# B&R Automation Studio project FileXplore
Automation Studio 6.7.0.187; technology packages: mappCockpit 6.6.0, mappView 6.6.0, OpcUaCs 6.6.1

## Configuration PLC

CPU X20CP3687X, AutomationRuntime 6.8.1, Build 11.3.0, Vc 6.0.0

### Task classes (Cpu.sw)
```
Cyclic#1:
  XFiles <- Source.XFiles.prg
Binaries: FWRules, ArSvcReg, TCData, udbdef, TCLang, mvLoader, mvConfig, User, iomap, TC, sysconf, BRRole, Role, arconfig, asfw, ashwac, Settings, UaCsConfig, ashwd, mCoWebSc
Libraries: runtime, AsZip, FileIO, AsHttp, UaCore, UaCoal, AsIecCon, ArSsl, UaCoalPrv, CoTrace, XFileLib, AsIODiag
```

### Hardware
```
X20CP3687X : X20CP3687X v1.9.0.0
  Connector IF2:
    ActivateDevice = 1
    Mode = Manual
    InternetAddress = 192.168.3.100
    SubnetMask = 255.255.255.0
    ActivateSnmp = 2
  ConfigurationID = FileXplore_PLC
  UserPartitionSize = 100
  Simulation = 1
  FileDevice1
  FileDeviceName1 = USER
  FileDevicePath1 = USER_PATH
  FileDevice2
  FileDeviceName2 = XPlore
  FileDevicePath2 = USER_PATH\XPlore
  ActivateFtpServer = 1
  FTPProtocol = 1
  FtpUser1
  FtpUsername1 = FileX
  FtpUserPassword1 = 8JF6nSqDfWDJ2i1aTp85XN0mfqkVcSXatZ/FMR942Jg=  // Password: XFile
  FtpUserSalt1 = RJsmGuSw
  FTPAccessRight1 = 0
  ActivateWebServer = 1
  WebServerProtocol = 3
  HttpsSslCfg = SSLConfiguration
  WebServerWebDir = dist\
```

## Logical view

Binary libraries used (declarations not repeated): operator, runtime, AsIecCon, AsZip, FileIO, AsHttp, CoTrace 6.5.0, AsIODiag

### Global.var - Global variables
```iecst
VAR
	gHostIP : STRING[15];
END_VAR
```


### Package Logical/FileXplore - File Xplorer source code (vite/react)

### CHANGELOG.md
```markdown
# Changelog

All notable changes to FileXplorer are documented here.

## [2.0.2] - 2026-10-08
- Added `ForceConvertToUTF8` config option: files whose extension is listed are converted to UTF-8 before transfer (BOM-aware, with Windows ANSI/CP1252 and UTF-16 fallback). An empty or missing list disables conversion.
- Added a Refresh button to reload the current folder without leaving it.
- Fixed the Home button doing nothing when already at the default path; it now always reloads.

## [2.0.1] - 2026-09-30
- FileXplore version shown only 1 second

## [2.0.0] - 2026-09-25

- Added a version display showing FileXplore for five seconds.
- Modified ftp to chunked HTTPS file uploads (works in arsim also)
- Added filename header sanitization for PLC-compatible transfers.
- Added configurable file browsing and transfer settings.
```

- package-lock.json (not shown)

- package.json (not shown)

### README.md
~~~~markdown
# File Explorer with HTTPS Transfer

A Vite + React file explorer application with Node.js backend designed for **B&R mappView environments**. The application enables browsing local files and transferring them to a PLC over chunked HTTPS, featuring real-time progress tracking and transfer recovery handling.

## Use Case

This application is intended to run in **B&R mappView** environments where:
- The **frontend** runs in the mappView HMI interface
- The **Node.js backend** runs on a **Panel PC** or another platform capable of accessing the local file system
- The **HTTPS endpoint** is a **B&R PLC** service that receives the selected files from the file explorer
- Files are streamed from the Panel PC (or host platform) to the PLC via bounded HTTPS chunks

## Features

### File Browsing
- Browse files and directories from configured drives on your local machine
- Tree-view navigation with expand/collapse folders
- Drive selection dropdown
- Configurable file extension filtering (e.g., `.txt`, `.cnc`)
- Access restrictions to prevent navigation outside configured directories

### HTTPS Transfer
- One-click file transfer to HTTPS endpoint (B&R PLC)
- Real-time upload progress tracking using Server-Sent Events (SSE)
- Visual progress bar showing actual HTTPS transfer percentage
- Transfer cancellation support (client and server-side)
- Configurable chunk size, timeout, and retry handling for transient transfer failures
- Automatic file load command trigger after successful upload to PLC
- Green highlight for successfully transferred files

### Configuration
- **Frontend Config** (`public/config.json`): Supported file extensions and default drive paths
- **Backend Config** (`server/https-config.json`): PLC HTTPS endpoint, chunk size, timeout, retry, default folder, and filename settings

## Project Structure

```
├── public/
│   └── config.json          # Frontend configuration
├── server/
│   ├── index.js             # Express backend server
│   └── https-config.json    # HTTPS transfer configuration
├── src/
│   ├── App.jsx              # Main React application
│   ├── App.css              # Application styles
│   └── main.jsx             # React entry point
└── dist/                    # Production build output
```

## Getting Started

### Backend Server (Panel PC or Host Platform)
The Node.js backend should run on a Panel PC or any platform with access to the local file system containing the files to be transferred.

```bash
cd server
node index.js
```
Server runs on `http://localhost:5000`

### Frontend (mappView HMI)
For development:
```bash
npm run dev
```
Development server runs on `http://localhost:5173`

### Production Build (for mappView deployment)
```bash
npm run build
node serve-dist.js
```
Serves production build on `http://localhost:3000`

The `dist` folder can be deployed to the mappView project.

## Running Backend as a Windows Service

To ensure the Node.js backend server runs automatically on PC startup and restarts after reboots, set it up as a Windows service.

### Option 1: Using node-windows (Recommended)

1. Install node-windows in the server directory:
```bash
cd server
npm install node-windows
```

2. Create a service installation script `install-service.js`:
```javascript
const Service = require('node-windows').Service;
const path = require('path');

// Create a new service object
const svc = new Service({
  name: 'FileExplorer Backend',
  description: 'File Explorer Node.js backend for B&R mappView',
  script: path.join(__dirname, 'index.js'),
  nodeOptions: [
    '--harmony',
    '--max_old_space_size=4096'
  ]
});

// Listen for the "install" event
svc.on('install', function() {
  svc.start();
  console.log('Service installed and started!');
});

// Install the service
svc.install();
```

3. Run the installation script as Administrator:
```bash
node install-service.js
```

4. To uninstall the service, create `uninstall-service.js`:
```javascript
const Service = require('node-windows').Service;
const path = require('path');

const svc = new Service({
  name: 'FileExplorer Backend',
  script: path.join(__dirname, 'index.js')
});

svc.on('uninstall', function() {
  console.log('Service uninstalled');
});

svc.uninstall();
```

### Option 2: Using Windows Task Scheduler

1. Open Task Scheduler (taskschd.msc)
2. Click "Create Task" (not "Create Basic Task")
3. **General tab**:
   - Name: "FileExplorer Backend"
   - Select "Run whether user is logged on or not"
   - Check "Run with highest privileges"
4. **Triggers tab**:
   - New → Begin the task: "At startup"
   - Delay task for: 30 seconds (to ensure network is ready)
5. **Actions tab**:
   - New → Action: "Start a program"
   - Program/script: `C:\Program Files\nodejs\node.exe`
   - Add arguments: `C:\path\to\your\server\index.js`
   - Start in: `C:\path\to\your\server`
6. **Conditions tab**:
   - Uncheck "Start the task only if the computer is on AC power"
7. Click OK and enter your Windows password

### Option 3: Using PM2 (Alternative)

1. Install PM2 globally:
```bash
npm install -g pm2
npm install -g pm2-windows-startup
```

2. Configure PM2 to start on boot:
```bash
pm2-startup install
```

3. Start your application with PM2:
```bash
cd server
pm2 start index.js --name "fileexplorer-backend"
pm2 save
```

### Verify Service is Running

Check if the service is running by accessing `http://localhost:5000/api/drives` in a browser or test it after a reboot.

## API Endpoints

- `GET /api/drives` - List available drives on the host platform
- `GET /api/list?path=<path>` - List directory contents from host file system
- `GET /api/read-file?path=<path>` - Read file as binary stream from host
- `POST /api/save-to-https-static` - Stream file from backend host to PLC HTTPS endpoint in chunks with progress (SSE)
- `POST /api/cancel-upload` - Cancel active HTTPS upload to PLC
- `POST /api/load-selected-file` - Trigger file load command on PLC

## Technologies

- **Frontend**: React 18, Vite, CSS (deployable to B&R mappView HTML )
- **Backend**: Node.js, Express (runs on Panel PC or host platform)
- **Transfer**: Node.js native HTTPS chunk upload client
- **Progress Tracking**: Server-Sent Events (SSE)
- **Target**: B&R PLC with HTTPS service capability
~~~~

- config.json (not shown)

- ftp-config.json (not shown)

### How to run.txt
```
1. Install node.js server (Chrome downloads)
2. Install Express via npm install express (from command line)
3. Install the node production process manager and run the node application (from command line):
	npm install -g pm2
	pm2 start app.js
	pm2 save
	pm2-startup install
```

- https-config.json (not shown)

- package-lock.json (not shown)

- package.json (not shown)

- App.jsx (not shown)

### Package Logical/Source - Source code for PLC code

### Library Logical/Source/XFileLib (IEC) - Library for file managment backend functionality

#### Types.typ - Exported data types
```iecst
TYPE
	XploreUploadStep_typ :
		(
		XPLORE_UPLOAD_IDLE := 0,
		XPLORE_UPLOAD_DELETE := 10,
		XPLORE_UPLOAD_CREATE := 20,
		XPLORE_UPLOAD_OPEN := 30,
		XPLORE_UPLOAD_WRITE := 40,
		XPLORE_UPLOAD_CLOSE := 50,
		XPLORE_UPLOAD_RESPOND := 60,
		XPLORE_UPLOAD_ERROR := 100
		);
	XploreHttpsServices_typ : 	STRUCT
		LoadServiceName : STRING[80];
		UploadServiceName : STRING[80];
		FileDevice : STRING[20];
		LoadRequestHeader : httpRequestHeader_t;
		LoadRequest : STRING[1000];
		LoadResponseHeader : httpResponseHeader_t;
		LoadResponse : STRING[1000];
		UploadRequestHeader : httpRequestHeader_t;
		UploadData : ARRAY[0..MAX_DATA_PAYLOAD_SIZE_BYTES]OF USINT;
		UploadResponseHeader : httpResponseHeader_t;
		UploadResponse : STRING[1000];
		FileName : STRING[80];
		TransferId : STRING[80];
		UploadOffset : UDINT;
		UploadLength : UDINT;
		UploadFileSize : UDINT;
		UploadChunkIndex : UDINT;
		UploadBytesReceived : UDINT;
		UploadStep : XploreUploadStep_typ;
		FileIdent : UDINT;
		Busy : BOOL;
		Done : BOOL;
		Error : BOOL;
		LastError : UINT;
		LastErrorText : STRING[80];
		LastHttpStatus : UINT;
		LastChunkFinal : BOOL;
		Reset : BOOL;
	END_STRUCT;
END_TYPE
```

#### Constants.var - Exported constants
```iecst
VAR CONSTANT
	MAX_DATA_PAYLOAD_SIZE_BYTES : UDINT := 1048576*MAX_DATA_PAYLOAD_SIZE_MB;
	MAX_DATA_PAYLOAD_SIZE_MB : UDINT := 5; (*This is the value to set for the file transfer*)
END_VAR
```

#### XFileLib.fun - Exported functions and function blocks
```iecst
{REDUND_ERROR} {REDUND_UNREPLICABLE} FUNCTION_BLOCK XploreFileService (*Xplore file service (HTTPS)*) (*$GROUP=User,$CAT=User,$GROUPICON=User.png,$CATICON=User.png*)
	VAR_INPUT
		Enable : {REDUND_UNREPLICABLE} BOOL;
		Reset : {REDUND_UNREPLICABLE} BOOL;
		FileDevice : {REDUND_UNREPLICABLE} STRING[20];
		LoadServiceName : {REDUND_UNREPLICABLE} STRING[80];
		UploadServiceName : {REDUND_UNREPLICABLE} STRING[80];
	END_VAR
	VAR_OUTPUT
		Busy : {REDUND_UNREPLICABLE} BOOL;
		Done : {REDUND_UNREPLICABLE} BOOL;
		Error : {REDUND_UNREPLICABLE} BOOL;
		FileName : {REDUND_UNREPLICABLE} STRING[80];
		UploadBytesReceived : {REDUND_UNREPLICABLE} UDINT;
		LastError : {REDUND_UNREPLICABLE} UINT;
		LastErrorText : {REDUND_UNREPLICABLE} STRING[80];
		LastHttpStatus : {REDUND_UNREPLICABLE} UINT;
	END_VAR
	VAR
		loadHttpsService : {REDUND_UNREPLICABLE} httpsService;
		uploadHttpsService : {REDUND_UNREPLICABLE} httpsService;
		fileDelete : {REDUND_UNREPLICABLE} FileDelete;
		fileCreate : {REDUND_UNREPLICABLE} FileCreate;
		fileOpen : {REDUND_UNREPLICABLE} FileOpen;
		fileWrite : {REDUND_UNREPLICABLE} FileWrite;
		fileClose : {REDUND_UNREPLICABLE} FileClose;
		service : {REDUND_UNREPLICABLE} XploreHttpsServices_typ;
	END_VAR
END_FUNCTION_BLOCK
```

#### XploreFileService.st - Reusable XFiles HTTP and file transfer service
```iecst
FUNCTION_BLOCK XploreFileService
	service.LoadServiceName := LoadServiceName;
	service.UploadServiceName := UploadServiceName;
	service.FileDevice := FileDevice;

	loadHttpsService(enable := Enable AND NOT Reset,
		option := httpOPTION_SERVICE_TYPE_NAME,
		pServiceName := ADR(service.LoadServiceName),
		pRequestHeader := ADR(service.LoadRequestHeader),
		pRequestData := ADR(service.LoadRequest),
		requestDataSize := SIZEOF(service.LoadRequest),
		pResponseHeader := ADR(service.LoadResponseHeader),
		pResponseData := ADR(service.LoadResponse),
		responseDataLen := SIZEOF(service.LoadResponse));
	uploadHttpsService(enable := Enable AND NOT Reset,
		option := httpOPTION_SERVICE_TYPE_NAME,
		pServiceName := ADR(service.UploadServiceName),
		pRequestHeader := ADR(service.UploadRequestHeader),
		pRequestData := ADR(service.UploadData),
		requestDataSize := SIZEOF(service.UploadData),
		pResponseHeader := ADR(service.UploadResponseHeader),
		pResponseData := ADR(service.UploadResponse),
		responseDataLen := SIZEOF(service.UploadResponse));

	IF service.LoadRequestHeader.userLine[0].name = '' THEN
		service.LoadRequestHeader.userLine[0].name := 'fileName';
		service.UploadRequestHeader.userLine[0].name := 'fileName';
		service.UploadRequestHeader.userLine[1].name := 'remotePath';
		service.UploadRequestHeader.userLine[2].name := 'transferId';
		service.UploadRequestHeader.userLine[3].name := 'chunkOffset';
		service.UploadRequestHeader.userLine[4].name := 'chunkIndex';
		service.UploadRequestHeader.userLine[5].name := 'fileSize';
		service.UploadRequestHeader.userLine[6].name := 'finalChunk';
	END_IF

	IF loadHttpsService.phase = httpPHASE_RECEIVED THEN
		IF service.LoadRequest = 'Load' THEN
			service.LoadResponseHeader.status := '200 OK';
			service.LoadResponseHeader.contentType := 'text/plain';
			service.LoadResponse := 'Loading';
			service.LoadRequest := '';
			loadHttpsService.send := TRUE;
		END_IF
		service.FileName := service.LoadRequestHeader.userLine[0].value;
	ELSE
		loadHttpsService.send := FALSE;
	END_IF

	IF Reset OR NOT Enable THEN
		service.UploadStep := XPLORE_UPLOAD_IDLE;
		service.Busy := FALSE;
		service.Done := FALSE;
		service.Error := FALSE;
		service.LastError := ERR_OK;
		service.FileIdent := 0;
		uploadHttpsService.send := FALSE;
	ELSE
		IF (uploadHttpsService.phase = httpPHASE_RECEIVED) AND (service.UploadStep = XPLORE_UPLOAD_IDLE) THEN
			service.FileName := service.UploadRequestHeader.userLine[0].value;
			service.TransferId := service.UploadRequestHeader.userLine[2].value;
			service.UploadOffset := STRING_TO_UDINT(service.UploadRequestHeader.userLine[3].value);
			service.UploadChunkIndex := STRING_TO_UDINT(service.UploadRequestHeader.userLine[4].value);
			service.UploadFileSize := STRING_TO_UDINT(service.UploadRequestHeader.userLine[5].value);
			service.LastChunkFinal := service.UploadRequestHeader.userLine[6].value = '1';
			service.UploadLength := uploadHttpsService.requestDataLen;
			service.Busy := TRUE;
			service.Done := FALSE;
			service.Error := FALSE;
			service.LastError := ERR_OK;
			service.LastErrorText := '';
			service.LastHttpStatus := 0;
			IF uploadHttpsService.method <> httpMETHOD_POST THEN
				service.LastHttpStatus := 405;
				service.UploadStep := XPLORE_UPLOAD_ERROR;
			ELSIF service.FileName = '' THEN
				service.LastHttpStatus := 400;
				service.UploadStep := XPLORE_UPLOAD_ERROR;
			ELSIF service.UploadLength >= SIZEOF(service.UploadData) THEN
				service.LastHttpStatus := 413;
				service.UploadStep := XPLORE_UPLOAD_ERROR;
			ELSIF service.UploadOffset = 0 THEN
				service.UploadStep := XPLORE_UPLOAD_DELETE;
			ELSE
				service.UploadStep := XPLORE_UPLOAD_OPEN;
			END_IF
		END_IF

		CASE service.UploadStep OF
			XPLORE_UPLOAD_IDLE:
				uploadHttpsService.send := FALSE;

			XPLORE_UPLOAD_DELETE:
				fileDelete(enable := TRUE, pDevice := ADR(service.FileDevice), pName := ADR(service.FileName));
				IF (fileDelete.status = ERR_OK) OR (fileDelete.status = fiERR_FILE_NOT_FOUND) THEN
					fileDelete(enable := FALSE);
					service.UploadStep := XPLORE_UPLOAD_CREATE;
				ELSIF fileDelete.status <> ERR_FUB_BUSY THEN
					service.LastError := fileDelete.status;
					service.LastErrorText := UDINT_TO_STRING(UINT_TO_UDINT(fileDelete.status));
					service.LastHttpStatus := 500;
					fileDelete(enable := FALSE);
					service.UploadStep := XPLORE_UPLOAD_ERROR;
				END_IF

			XPLORE_UPLOAD_CREATE:
				fileCreate(enable := TRUE, pDevice := ADR(service.FileDevice), pFile := ADR(service.FileName));
				IF fileCreate.status = ERR_OK THEN
					service.FileIdent := fileCreate.ident;
					fileCreate(enable := FALSE);
					service.UploadStep := XPLORE_UPLOAD_WRITE;
				ELSIF fileCreate.status <> ERR_FUB_BUSY THEN
					service.LastError := fileCreate.status;
					service.LastErrorText := UDINT_TO_STRING(UINT_TO_UDINT(fileCreate.status));
					service.LastHttpStatus := 500;
					fileCreate(enable := FALSE);
					service.UploadStep := XPLORE_UPLOAD_ERROR;
				END_IF

			XPLORE_UPLOAD_OPEN:
				fileOpen(enable := TRUE, pDevice := ADR(service.FileDevice), pFile := ADR(service.FileName), mode := fiREAD_WRITE);
				IF fileOpen.status = ERR_OK THEN
					service.FileIdent := fileOpen.ident;
					fileOpen(enable := FALSE);
					service.UploadStep := XPLORE_UPLOAD_WRITE;
				ELSIF fileOpen.status <> ERR_FUB_BUSY THEN
					service.LastError := fileOpen.status;
					service.LastErrorText := UDINT_TO_STRING(UINT_TO_UDINT(fileOpen.status));
					service.LastHttpStatus := 409;
					fileOpen(enable := FALSE);
					service.UploadStep := XPLORE_UPLOAD_ERROR;
				END_IF

			XPLORE_UPLOAD_WRITE:
				fileWrite(enable := TRUE, ident := service.FileIdent, offset := service.UploadOffset, pSrc := ADR(service.UploadData), len := service.UploadLength);
				IF fileWrite.status = ERR_OK THEN
					fileWrite(enable := FALSE);
					service.UploadStep := XPLORE_UPLOAD_CLOSE;
				ELSIF fileWrite.status <> ERR_FUB_BUSY THEN
					service.LastError := fileWrite.status;
					service.LastErrorText := UDINT_TO_STRING(UINT_TO_UDINT(fileWrite.status));
					service.LastHttpStatus := 500;
					fileWrite(enable := FALSE);
					service.UploadStep := XPLORE_UPLOAD_CLOSE;
				END_IF

			XPLORE_UPLOAD_CLOSE:
				fileClose(enable := TRUE, ident := service.FileIdent);
				IF fileClose.status = ERR_OK THEN
					fileClose(enable := FALSE);
					service.FileIdent := 0;
					IF service.LastError = ERR_OK THEN
						service.UploadStep := XPLORE_UPLOAD_RESPOND;
					ELSE
						service.UploadStep := XPLORE_UPLOAD_ERROR;
					END_IF
				ELSIF fileClose.status <> ERR_FUB_BUSY THEN
					service.LastError := fileClose.status;
					service.LastErrorText := UDINT_TO_STRING(UINT_TO_UDINT(fileClose.status));
					service.LastHttpStatus := 500;
					fileClose(enable := FALSE);
					service.FileIdent := 0;
					service.UploadStep := XPLORE_UPLOAD_ERROR;
				END_IF

			XPLORE_UPLOAD_RESPOND:
				service.UploadBytesReceived := service.UploadOffset + service.UploadLength;
				service.UploadResponseHeader.status := '200 OK';
				service.UploadResponseHeader.contentType := 'text/plain';
				service.UploadResponse := 'OK';
				service.Done := service.LastChunkFinal;
				service.Busy := FALSE;
				uploadHttpsService.send := TRUE;
				service.UploadStep := XPLORE_UPLOAD_IDLE;

			XPLORE_UPLOAD_ERROR:
				service.Error := TRUE;
				service.Busy := FALSE;
				IF service.LastHttpStatus = 0 THEN
					service.LastHttpStatus := 500;
				END_IF
				IF service.LastHttpStatus = 400 THEN
					service.UploadResponseHeader.status := '400 Bad Request';
				ELSIF service.LastHttpStatus = 405 THEN
					service.UploadResponseHeader.status := '405 Method Not Allowed';
				ELSIF service.LastHttpStatus = 409 THEN
					service.UploadResponseHeader.status := '409 Conflict';
				ELSIF service.LastHttpStatus = 413 THEN
					service.UploadResponseHeader.status := '413 Payload Too Large';
				ELSE
					service.UploadResponseHeader.status := '500 Internal Server Error';
				END_IF
				service.UploadResponseHeader.contentType := 'text/plain';
				service.UploadResponse := service.LastErrorText;
				uploadHttpsService.send := TRUE;
				service.UploadStep := XPLORE_UPLOAD_IDLE;
		END_CASE
	END_IF

	Busy := service.Busy;
	Done := service.Done;
	Error := service.Error;
	FileName := service.FileName;
	UploadBytesReceived := service.UploadBytesReceived;
	LastError := service.LastError;
	LastErrorText := service.LastErrorText;
	LastHttpStatus := service.LastHttpStatus;
END_FUNCTION_BLOCK
```

### Program Logical/Source/XFiles (IEC) -  Sample code to get the selected files from FileXplorer

#### Types.typ
```iecst
TYPE
	XploreUploadStep_typ :
		(
			XPLORE_UPLOAD_IDLE := 0,
			XPLORE_UPLOAD_DELETE := 10,
			XPLORE_UPLOAD_CREATE := 20,
			XPLORE_UPLOAD_OPEN := 30,
			XPLORE_UPLOAD_WRITE := 40,
			XPLORE_UPLOAD_CLOSE := 50,
			XPLORE_UPLOAD_RESPOND := 60,
			XPLORE_UPLOAD_ERROR := 100
		);

	XploreHttpServices_typ : 	STRUCT
		LoadServiceName : STRING[80];
		UploadServiceName : STRING[80];
		FileDevice : STRING[20];
		LoadRequestHeader : httpRequestHeader_t;
		LoadRequest : STRING[1000];
		LoadResponseHeader : httpResponseHeader_t;
		LoadResponse : STRING[1000];
		UploadRequestHeader : httpRequestHeader_t;
		UploadData : ARRAY[0..32767] OF USINT;
		UploadResponseHeader : httpResponseHeader_t;
		UploadResponse : STRING[1000];
		FileName : STRING[80];
		TransferId : STRING[80];
		UploadOffset : UDINT;
		UploadLength : UDINT;
		UploadFileSize : UDINT;
		UploadChunkIndex : UDINT;
		UploadBytesReceived : UDINT;
		UploadStep : XploreUploadStep_typ;
		FileIdent : UDINT;
		Busy : BOOL;
		Done : BOOL;
		Error : BOOL;
		LastError : UINT;
		LastErrorText : STRING[80];
		LastHttpStatus : UINT;
		LastChunkFinal : BOOL;
		Reset : BOOL;
	END_STRUCT;
END_TYPE
```

#### Variables.var
```iecst
VAR
	cpuSimulated : BOOL;
	xploreFileService_0 : XploreFileService;
END_VAR
```

#### Main.st
```iecst
PROGRAM _INIT
	xploreFileService_0(
		Enable := FALSE,
		Reset := TRUE,
		FileDevice := 'XPlore',
		LoadServiceName := 'load-selected-Xfile',
		UploadServiceName := 'upload-Xfile');

		cpuSimulated := DiagCpuIsARsim();
END_PROGRAM

PROGRAM _CYCLIC
	xploreFileService_0(
		Enable := TRUE,
		Reset := FALSE,
		FileDevice := 'XPlore',
		LoadServiceName := 'load-selected-Xfile',
		UploadServiceName := 'upload-Xfile');

		IF cpuSimulated THEN
			gHostIP := '127.0.0.1'; //Simulation active
		ELSE
			gHostIP := '192.168.3.100'; //Real target
		END_IF

END_PROGRAM

PROGRAM _EXIT
	xploreFileService_0(
		Enable := FALSE,
		Reset := TRUE,
		FileDevice := 'XPlore',
		LoadServiceName := 'load-selected-Xfile',
		UploadServiceName := 'upload-Xfile');
END_PROGRAM
```

- Visualisation Logical/mappView (not shown)

Listed in the project but not available here: Logical/Global.typ
